(* IEC 61131-3 sources: InfiniteStateMachine/extracted_st/infinitestatemachine/globalconstants/ism, 1 file *)

(* ---- ISM.st ---- *)
(* --- Interface --- *)
{attribute 'qualified_only'}
VAR_GLOBAL CONSTANT
	gc_iMaxDepth : INT := 7;
END_VAR
